FUNCTION_BLOCK A2X2_2X_TO_2AX2 (* Composite FB for convert A2X2 to 2 AX2 *)
  (* Standard: 61499-2; Description: Copyright (c) 2026 HR Agrartechnik GmbH This program and the accompanying materials are made available under the terms of the Eclipse Public License 2.0 which is available at https://www.eclipse.org/legal/epl-2.0/ SPDX-License-Identifier: EPL-2.0 *)
  (* Version 1.0, 2026-08-31, Franz Höpfinger, HR Agrartechnik GmbH *)
  PACKAGE adapter::conversion::bidirectional;
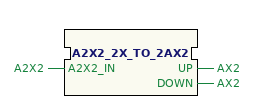
  SOCKETS
    A2X2_IN : adapter::types::bidirectional::A2X2; (* Adapter Input *)
  END_SOCKETS
  PLUGS
    UP : adapter::types::bidirectional::AX2; (* TRUE = forward, up, right, clockwise *)
    DOWN : adapter::types::bidirectional::AX2; (* TRUE = backward, down, left, counter-clockwise *)
  END_PLUGS
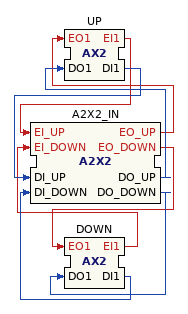
  EVENT_CONNECTIONS
    A2X2_IN.EO_UP TO UP.EO1;
    UP.EI1 TO A2X2_IN.EI_UP;
    A2X2_IN.EO_DOWN TO DOWN.EO1;
    DOWN.EI1 TO A2X2_IN.EI_DOWN;
  END_CONNECTIONS
  DATA_CONNECTIONS
    A2X2_IN.DO_UP TO UP.DO1;
    UP.DI1 TO A2X2_IN.DI_UP;
    A2X2_IN.DO_DOWN TO DOWN.DO1;
    DOWN.DI1 TO A2X2_IN.DI_DOWN;
  END_CONNECTIONS
END_FUNCTION_BLOCK
